(* IEC 61131-3 sources: CodesysTest/alpha/export/FBs/Fault/FB_Fault.pou/InstanceName.prop, 1 file *)

(* ---- Get.pm.st ---- *)
(*#-#-#-#-#-#-#-#-#-#---Declaration---#-#-#-#-#-#-#-#-#-#-#-#-#*)

VAR
END_VAR
(*#-#-#-#-#-#-#-#-#-#---Implementation---#-#-#-#-#-#-#-#-#-#-#-#-#*)

InstanceName := _instanceName;
